KUKA KRL program: krl_test.src, krl_test.dat

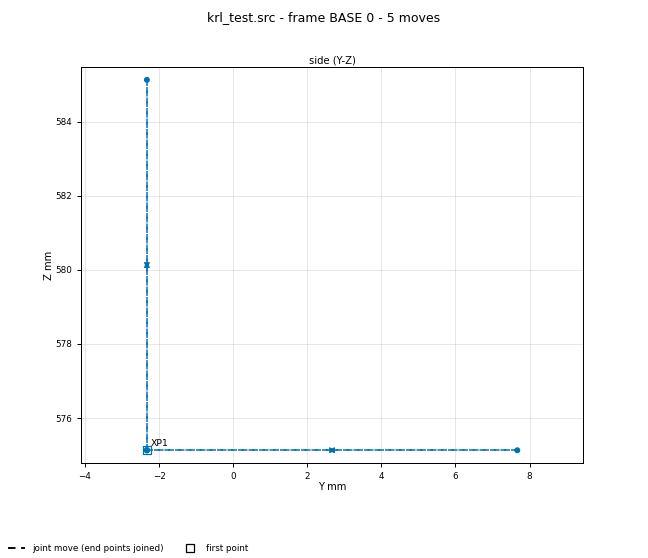
[picture p0: tool path of krl_test.src in frame BASE 0, 5 of 5 moves have a stored position in this frame; points joined in program order, loops and branches not executed]
--- krl_test.src ---
&ACCESS RVP
&REL 13
&PARAM EDITMASK = *
&PARAM TEMPLATE = C:\KRC\Roboter\Template\vorgabe
&PARAM DISKPATH = KRC:\R1\Program
DEF krl_test( )
;FOLD Declaration
  DECL EKI_STATUS RET
  INT OFFSET
  REAL ind
  INT Counter
  BOOL valueBool
  INT i
  REAL valueReal
  CHAR Bytes[4]
  FOR i=(1) TO (4)
     Bytes[i]=0
  ENDFOR
  OFFSET=0
  Counter=0
  ind=0.0
;ENDFOLD (Declaration)

;FOLD INI;%{PE}
  ;FOLD BASISTECH INI
    GLOBAL INTERRUPT DECL 3 WHEN $STOPMESS==TRUE DO IR_STOPM ( )
    INTERRUPT ON 3
    BAS (#INITMOV,0 )
  ;ENDFOLD (BASISTECH INI)
  ;FOLD USER INI
    ;Make your modifications here

  ;ENDFOLD (USER INI)
;ENDFOLD (INI)

RET=EKI_Init("XmlServer")
RET=EKI_Open("XmlServer")

;FOLD SPTP P3 Vel=50 % PDAT3 Tool[1]:SMC Base[0] ;%{PE}
;FOLD Parameters ;%{h}
;Params IlfProvider=kukaroboter.basistech.inlineforms.movement.spline; Kuka.IsGlobalPoint=False; Kuka.PointName=P3; Kuka.BlendingEnabled=False; Kuka.MoveDataPtpName=PDAT3; Kuka.VelocityPtp=50; Kuka.VelocityFieldEnabled=True; Kuka.ColDetectFieldEnabled=True; Kuka.CurrentCDSetIndex=0; Kuka.MovementParameterFieldEnabled=True; IlfCommand=SPTP
;ENDFOLD
SPTP XP1 WITH $VEL_AXIS[1] = SVEL_JOINT(50.0), $TOOL = STOOL2(FP1), $BASE = SBASE(FP1.BASE_NO), $IPO_MODE = SIPO_MODE(FP1.IPO_FRAME), $LOAD = SLOAD(FP1.TOOL_NO), $ACC_AXIS[1] = SACC_JOINT(PPDAT1), $APO = SAPO_PTP(PPDAT1), $GEAR_JERK[1] = SGEAR_JERK(PPDAT1), $COLLMON_TOL_PRO[1] = USE_CM_PRO_VALUES(0)
;ENDFOLD
; wait until server is conntected
REPEAT
    wait for $FLAG[1]
    REPEAT
    RET=EKI_GetString("XmlServer","number",Bytes[])
    UNTIL (RET.Buff < 1)
    OFFSET=0
    CAST_FROM(Bytes[],OFFSET,valueReal)
    Counter=Counter+1
    IF valueReal == 1 THEN
       PTP_REL {Z 10}
    ENDIF
    IF valueReal == 2 THEN

       PTP_REL {Z -10}
    ENDIF
    IF valueReal == 3 THEN
       PTP_REL {Y 10}
    ENDIF
    IF valueReal == 4 THEN
       PTP_REL {Y -10}
    ENDIF
UNTIL (Counter > 10)
IF valueReal >0 THEN
    valueBool=TRUE

ENDIF




wait for valueBool
; wait until server is deconnected
wait for $FLAG[1]==FALSE

RET=EKI_Clear("XmlServer")
END

--- krl_test.dat ---
&ACCESS RVP
&REL 13
&PARAM EDITMASK = *
&PARAM TEMPLATE = C:\KRC\Roboter\Template\vorgabe
&PARAM DISKPATH = KRC:\R1\Program
DEFDAT  KRL_TEST
;FOLD EXTERNAL DECLARATIONS;%{PE}%MKUKATPBASIS,%CEXT,%VCOMMON,%P
;FOLD BASISTECH EXT;%{PE}%MKUKATPBASIS,%CEXT,%VEXT,%P
EXT  BAS (BAS_COMMAND  :IN,REAL  :IN )
DECL INT SUCCESS
;ENDFOLD (BASISTECH EXT)
;FOLD USER EXT;%{E}%MKUKATPUSER,%CEXT,%VEXT,%P
;Make your modifications here

;ENDFOLD (USER EXT)
;ENDFOLD (EXTERNAL DECLARATIONS)
DECL E6POS XP1={X 440.626801,Y -2.33104324,Z 575.130310,A 6.41748920E-05,B 89.8853531,C 0.00500106765,S 2,T 43,E1 0.0,E2 0.0,E3 0.0,E4 0.0,E5 0.0,E6 0.0}
DECL FDAT FP1={TOOL_NO 1,BASE_NO 0,IPO_FRAME #BASE,POINT2[] " "}
DECL PDAT PPDAT1={VEL 50.0000,ACC 100.000,APO_DIST 500.000,APO_MODE #CDIS,GEAR_JERK 100.000,EXAX_IGN 0}
DECL MODULEPARAM_T LAST_TP_PARAMS={PARAMS[] "Kuka.VelocityFieldEnabled=False; Kuka.ColDetectFieldEnabled=False; Kuka.MovementParameterFieldEnabled=False; Kuka.IsAngleEnabled=False; Kuka.PointName=P1; Kuka.FrameData.base_no=0; Kuka.FrameData.tool_no=1; Kuka.FrameData.ipo_frame=#BASE; Kuka.isglobalpoint=False; Kuka.MoveDataPtpName=PDAT1; Kuka.MovementDataPdat.apo_mode=#CDIS; Kuka.MovementDataPdat.apo_dist=500; Kuka.MovementData.vel=50; Kuka.MovementData.acc=100; Kuka.MovementData.gear_jerk=100; Kuka.MovementData.exax_ign=0; Kuka.VelocityPtp=50; Kuka.BlendingEnabled=False; Kuka.CurrentCDSetIndex=0"}
DECL E6POS XP2={X 440.626801,Y -2.33104324,Z 575.130310,A 6.41748920E-05,B 89.8853531,C 0.00500106765,S 2,T 43,E1 0.0,E2 0.0,E3 0.0,E4 0.0,E5 0.0,E6 0.0}
DECL FDAT FP2={TOOL_NO 1,BASE_NO 0,IPO_FRAME #BASE,POINT2[] " "}
DECL PDAT PPDAT2={VEL 50.0000,ACC 100.000,APO_DIST 500.000,APO_MODE #CDIS,GEAR_JERK 100.000,EXAX_IGN 0}
DECL E6POS XP3={X 440.626801,Y -2.33104324,Z 575.130310,A 6.41748920E-05,B 89.8853531,C 0.00500106765,S 2,T 43,E1 0.0,E2 0.0,E3 0.0,E4 0.0,E5 0.0,E6 0.0}
DECL FDAT FP3={TOOL_NO 1,BASE_NO 0,IPO_FRAME #BASE,POINT2[] " "}
DECL PDAT PPDAT3={VEL 50.0000,ACC 100.000,APO_DIST 500.000,APO_MODE #CDIS,GEAR_JERK 100.000,EXAX_IGN 0}
ENDDAT
